{attribute 'Tc2GvlVarNames'}
VAR_GLOBAL CONSTANT
	(* System_WDT_Zustand_Status *)
	E_System_WDT_Zustand_Status_Idle_Sperre				: SINT := 0;
	E_System_WDT_Zustand_Status_Betriebsbereit			: SINT := 1;
	E_System_WDT_Zustand_Status_Nachl_Stellventil		: SINT := 2;
	E_System_WDT_Zustand_Status_Vorl_Stellventil		: SINT := 3;
	E_System_WDT_Zustand_Status_Nachl_Pumpe				: SINT := 4;
	E_System_WDT_Zustand_Status_Vorl_Pumpe				: SINT := 5;
	E_System_WDT_Zustand_Status_Nachl_Regelventil		: SINT := 6;
	E_System_WDT_Zustand_Status_Vorl_Regelventil		: SINT := 7;
	E_System_WDT_Zustand_Status_Betrieb					: SINT := 8;
	E_System_WDT_Zustand_Status_Betrieb_Sperre			: SINT := 9;
	E_System_WDT_Zustand_Status_Stoerung				: SINT := 99;

	(* System_WDT_Zustand_Regelung_Modus *)
	E_System_WDT_Regelung_Modus_Automatik						: SINT := 0;
	E_System_WDT_Regelung_Modus_Heizen_viaNetz_konst			: SINT := 1;
	E_System_WDT_Regelung_Modus_Heizen_viaNetz_Kurve			: SINT := 2;
	E_System_WDT_Regelung_Modus_Heizen_viaRueckkuehler_konst	: SINT := 3;
	E_System_WDT_Regelung_Modus_Heizen_viaRueckkuehler_Kurve	: SINT := 4;
	E_System_WDT_Regelung_Modus_Kuehlen_viaNetz_konst			: SINT := -1;
	E_System_WDT_Regelung_Modus_Kuehlen_viaNetz_Kurve			: SINT := -2;
	E_System_WDT_Regelung_Modus_Kuehlen_viaRueckkuehler_konst	: SINT := -3;
	E_System_WDT_Regelung_Modus_Kuehlen_viaRueckkuehler_Kurve	: SINT := -4;
END_VAR

(* stored: Version 1.1.0.1, ProductVersion 3.1.4024.9
   GVL Con_WDT: Id {53abe389-a2a2-439a-b99b-b36aa18ade87} *)
